TYPE ST_POINTS :
STRUCT
	x : REAL;
	y : REAL;
END_STRUCT
END_TYPE

(* stored: Version 1.1.0.1, ProductVersion 3.1.4026.17
   DUT ST_POINTS: Id {f11cafda-f3e6-406e-b721-2282ef9985a8} *)
